(* CODESYS project BoxWrapper.project

Project tree, tasks and I/O mapping:
  Device : CODESYS Control Win V3 x64, 3S - Smart Software Solutions GmbH, version 3.5.12.10
    application Application
      libraries: Standard, * (System); VisuDialogs, * (System)
      task MainTask (cyclic, interval t#20ms, priority 1) calls PLC_PRG
      task VISU_TASK (cyclic, interval 100 ms, priority 31) calls VisuElems.Visu_Prg
      program PLC_PRG [LD]: Animation
      visualisation Box_Movement
  visualisation Box_movement
  text list GlobalTextList
*)

// Device/Application/PLC_PRG
PROGRAM PLC_PRG
VAR
	Start: BOOL;
	Stop: BOOL; 
	EMGC: BOOL;
	
	Rotation_coil: 				BOOL;
	Rotation_Frequency: 		INT;
	Rotation_OVLD: 				BOOL;
	
	Motor_Up_coil: 				BOOL;
	Motor_down_coil: 			BOOL;
	Motor_up_down_frequency: 	INT;
	Motor_up_down_OVLD: 		BOOL;
	
	
	Rotation_PX:				BOOL;
	Stretch_PX:					BOOL;
	
	HLMSW:						BOOL;
	LLMSW:						BOOL;
	
	Slider_low_count:			CTU;
	Slider_high_count:			CTU;
	
	
	
	
	UpBlinker: TON;
	DownBlinker: TON;
	UpDwoncounter: ctud;
	Rotation: TON;
	SliderCount: WORD;
	SliderAnimation: UINT;
	RotatoinCounter: CTU;
	RotationCounter: CTU;
	RotatoinCount: WORD;
	Rotation_Factor: INT;
	Rotation_Factro: INT;
	Motor_up_down_frequency_Factor: INT;
	Slider: UINT;
END_VAR
VAR // added by the converter: edge detectors and wires of the graphical bodies
    _rt1, _rt2, _rt3, _rt4 : R_TRIG;
    _ft1 : F_TRIG;
END_VAR

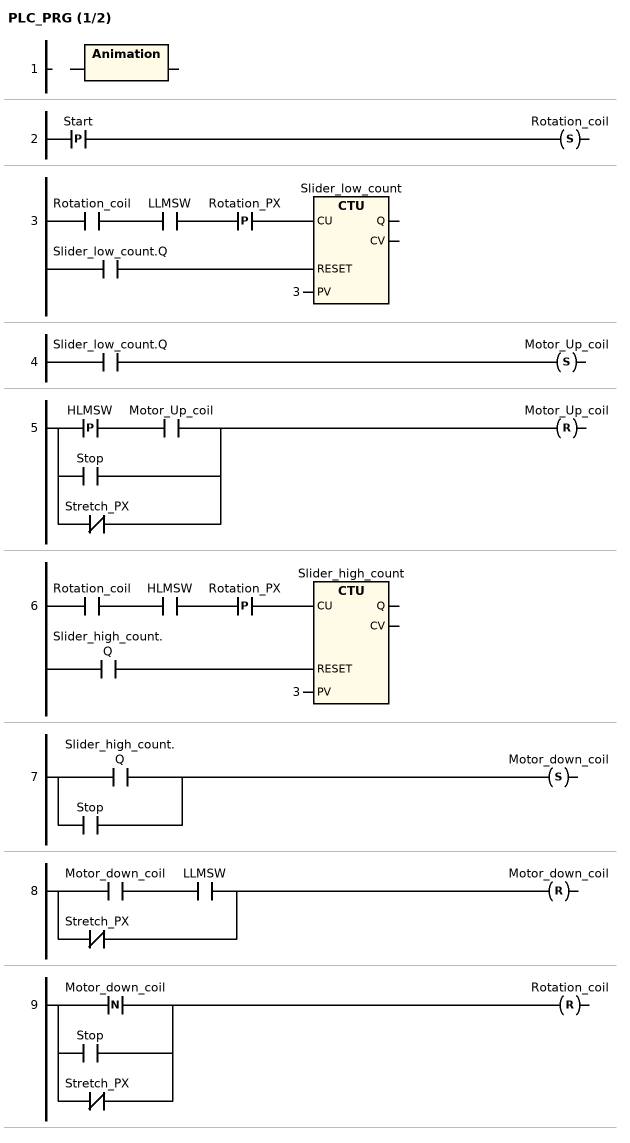
// NETWORK 1
Animation();

// NETWORK 2
_rt1(CLK := Start);
Rotation_coil S= _rt1.Q;

// NETWORK 3
_rt2(CLK := Rotation_PX);
Slider_low_count(CU := Rotation_coil AND LLMSW AND _rt2.Q, RESET := Slider_low_count.Q, PV := 3); // CTU

// NETWORK 4
Motor_Up_coil S= Slider_low_count.Q;

// NETWORK 5
_rt3(CLK := HLMSW);
Motor_Up_coil R= _rt3.Q AND Motor_Up_coil OR Stop OR NOT Stretch_PX;

// NETWORK 6
_rt4(CLK := Rotation_PX);
Slider_high_count(CU := Rotation_coil AND HLMSW AND _rt4.Q, RESET := Slider_high_count.Q, PV := 3); // CTU

// NETWORK 7
Motor_down_coil S= Slider_high_count.Q OR Stop;

// NETWORK 8
Motor_down_coil R= Motor_down_coil AND LLMSW OR NOT Stretch_PX;

// NETWORK 9
_ft1(CLK := Motor_down_coil);
Rotation_coil R= _ft1.Q OR Stop OR NOT Stretch_PX;

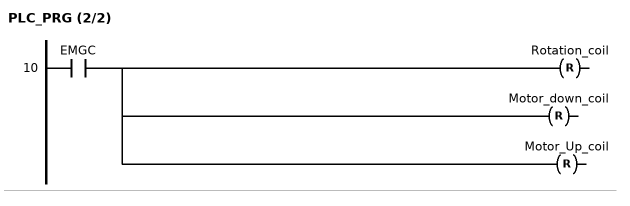
// NETWORK 10
Rotation_coil R= EMGC;
Motor_down_coil R= EMGC;
Motor_Up_coil R= EMGC;

ACTION Animation:
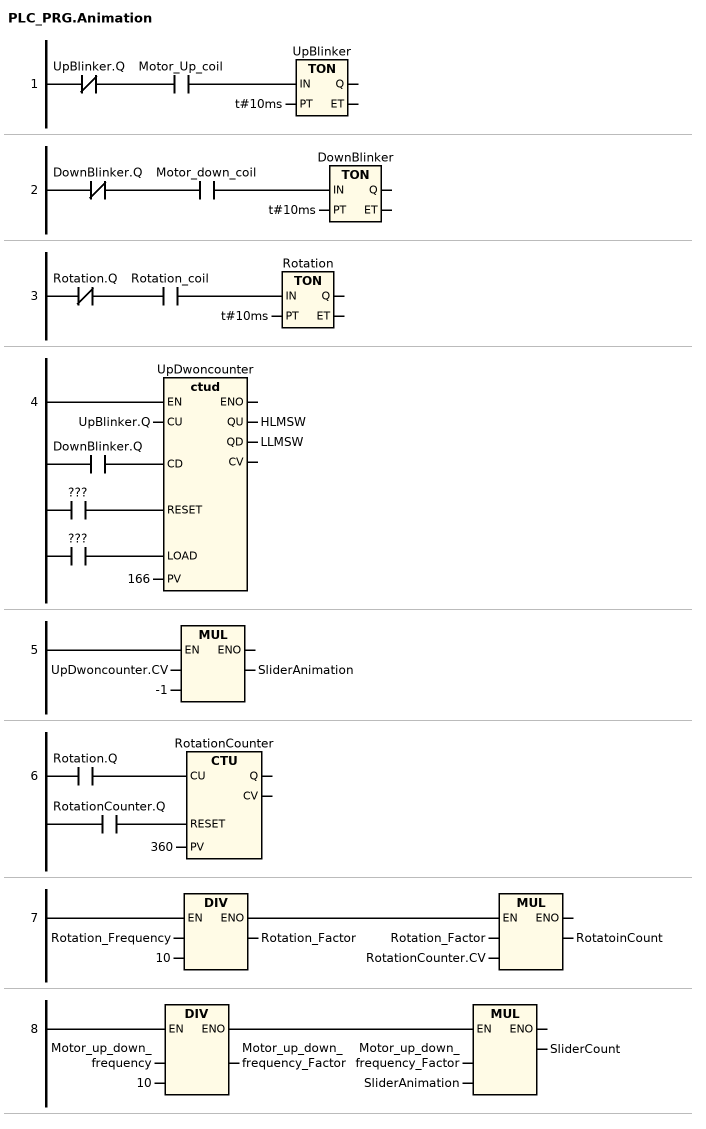
// NETWORK 1
UpBlinker(IN := NOT UpBlinker.Q AND Motor_Up_coil, PT := t#10ms); // TON

// NETWORK 2
DownBlinker(IN := NOT DownBlinker.Q AND Motor_down_coil, PT := t#10ms); // TON

// NETWORK 3
Rotation(IN := NOT Rotation.Q AND Rotation_coil, PT := t#10ms); // TON

// NETWORK 4
UpDwoncounter(CU := UpBlinker.Q, CD := DownBlinker.Q, PV := 166, QU => HLMSW, QD => LLMSW); // ctud

// NETWORK 5
SliderAnimation := UpDwoncounter.CV * -1;

// NETWORK 6
RotationCounter(CU := Rotation.Q, RESET := RotationCounter.Q, PV := 360); // CTU

// NETWORK 7
Rotation_Factor := Rotation_Frequency / 10;
RotatoinCount := Rotation_Factor * RotationCounter.CV;

// NETWORK 8
Motor_up_down_frequency_Factor := Motor_up_down_frequency / 10;
SliderCount := Motor_up_down_frequency_Factor * SliderAnimation;
END_ACTION

END_PROGRAM

// /Box_movement
VISUALIZATION Box_movement  // 2x2
END_VISUALIZATION

// Device/Application/Box_Movement
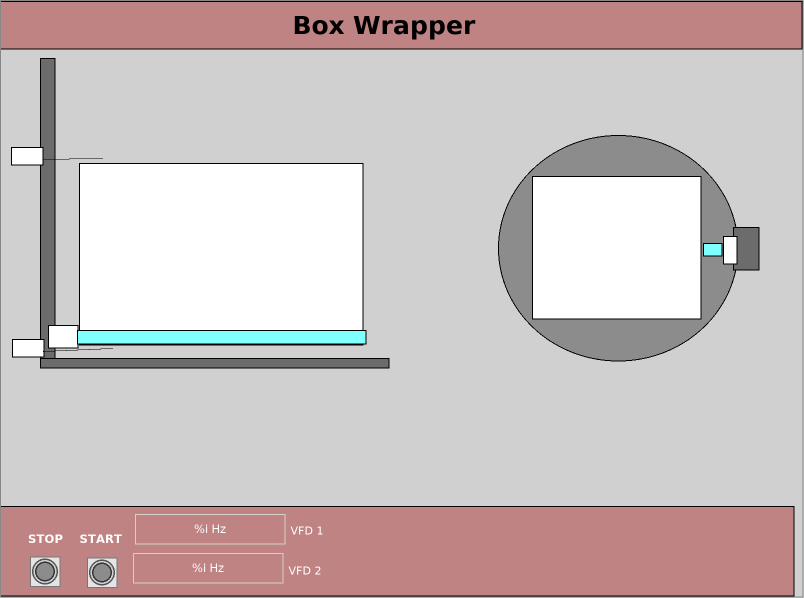
VISUALIZATION Box_Movement  // 804x598
    Rectangle (40,58 15x301)
    RoundedRectangle (40,358 349x10)
    Rectangle (79,163 284x182)
    Group (48,325 318x23)
        p2738717112: PLC_PRG.SliderCount
        Rectangle (0,0 30x23)
        RoundedRectangle (29,5 289x14)
    Ellipse (498,135 240x226)
    Rectangle (532,176 169x143)
        p2858320360: PLC_PRG.RotatoinCount
    Rectangle (733,227 26x43)
    Rectangle (723,236 14x28)
    RoundedRectangle (703,243 19x13)
    RoundedRectangle (-2,506 796x90)
    PushSwitch (30,550 30x43), variable: PLC_PRG.Stop, behaviour: TAP, style: Switch-PushSwitch-Gray
    PushSwitch (87,551 30x43), variable: PLC_PRG.Start, behaviour: TAP, style: Switch-PushSwitch-Gray
    Label (26,524 150x30), "START"
    Label (14,524 63x30), "STOP"
    Label (232,516 150x30), "VFD 1"
    Label (230,556 150x30), "VFD 2"
    Group (12,339 100x18)
        Rectangle (0,0 32x18)
        Line (31,12) (100,9)
    Group (11,147 91x18)
        Line (25,12) (91,11)
        Rectangle (0,0 32x18)
    Textfield (135,514 150x30), "%i Hz", text variable: PLC_PRG.Motor_up_down_frequency
        OnMouseClick: write the text variable via Default, min 0, max 50
    Textfield (133,553 150x30), "%i Hz", text variable: PLC_PRG.Rotation_Frequency
        OnMouseClick: write the text variable via Default, min 0, max 50
    RoundedRectangle (0,1 802x48)
    Label (260,10 248x30), "Box Wrapper"
END_VISUALIZATION
